// TIA Portal V17 program export: 0 tag tables, 0 data types, 0 data blocks, 2 code blocks (in call order from the OBs), 7 instance data blocks

ORGANIZATION_BLOCK "Main"   // OB1, LAD, ProgramCycle
TITLE = "Main Program Sweep (Cycle)"
{ S7_Optimized_Access := 'TRUE' }
VERSION : 0.1
// stored: AutoNumber true, IsIECCheckEnabled false, SetENOAutomatically false
   VAR_INPUT
      Initial_Call : Bool;   // Initial call of this OB
      Remanence : Bool;   // =True, if remanent data are available
   END_VAR
BEGIN

REGION Network 1
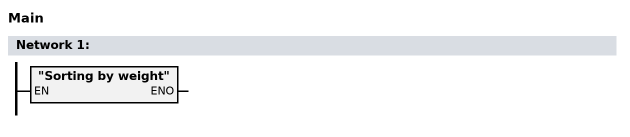
   RUNG wire#powerrail
      "Sorting by weight"()
   END_RUNG
   // the same network as SCL:
   "Sorting by weight"();
END_REGION
END_ORGANIZATION_BLOCK

FUNCTION "Sorting by weight" : Void
{ S7_Optimized_Access := 'TRUE' }
VERSION : 0.1

BEGIN
	IF "Start_PB" THEN
	    "MainConveyor" := TRUE;
	    "LeftConveyor" := TRUE;
	    "MiddleConveyor" := TRUE;
	    "RightConveyor" := TRUE;
	
	END_IF;
	
	
	"IEC_Timer_0_DB".TOF(IN:=NOT "Stop_Sensor",
	                     PT:=T#1S);
	"F_TRIG_DB"(CLK:="IEC_Timer_0_DB".Q);
	
	"IEC_Timer_0_DB_1".TOF(IN:=NOT "Stop_Sensor",
	                       PT:=T#3S);
	"F_TRIG_DB_1"(CLK:="IEC_Timer_0_DB_1".Q);
	
	
	IF "F_TRIG_DB".Q THEN
	    "ConveyorScale" := FALSE;
	ELSIF NOT "Stop_Sensor" THEN
	    "ConveyorScale" := TRUE;
	ELSIF "F_TRIG_DB_1".Q THEN
	    "ConveyorScale" := TRUE;
	END_IF;
	
	
	// Scaling of weight
	"Actual Weight":="ConveyorScaleWight"*2.0;
	
	
	//compare weight and respective data register
	IF NOT "ConveyorScale" AND "Actual Weight" >= 8.0 AND "Actual Weight" <= 8.2 THEN
	    "SortBIT" := 1;
	ELSIF NOT "ConveyorScale" AND "Actual Weight" >= 10.0 AND "Actual Weight" <= 10.2 THEN
	    "SortBIT" := 2;
	ELSIF NOT "ConveyorScale" AND "Actual Weight" > 15.0   THEN
	    "SortBIT" := 3;
	END_IF;
	
	
	// sort forward 10kg box
	IF "SortBIT"=2 THEN
	    "SortForword" := true;
	END_IF;
	
	// Reset forward sorting
	IF NOT "ExitSensorMiddle" THEN
	    "SortForword" := FALSE;
	    "SortLeft" := FALSE;
	    "SortRight" := FALSE;
	    "SortBIT" := 0;
	    "ConveyorScale" := FALSE;
	END_IF;
	
	
	// sort left 8kg box
	IF "SortBIT" = 1 THEN
	    "SortForword" := true;
	    "SortLeft" := true;
	END_IF;
	
	//reset left sorting
	IF NOT "ExitSensorLeft" THEN
	    "SortForword" := FALSE;
	    "SortLeft" := FALSE;
	    "SortRight" := FALSE;
	    "SortBIT" := 0;
	    "ConveyorScale" := 0;
	END_IF;
	
	
	// Sort right 15kg box
	IF "SortBIT" = 3 THEN
	    "SortForword" := true;
	    "SortRight" := true;
	END_IF;
	
	//reset right sorting 
	IF NOT "ExitSensorRight" THEN
	    "SortForword" := FALSE;
	    "SortLeft" := FALSE;
	    "SortRight" := FALSE;
	    "SortBIT" := 0;
	    "ConveyorScale" := 0;
	END_IF;
	
	
	// RESET ALL OUTPUT, MEMORY BIT , AND DATA REGISTER
	IF "Reset_PB" THEN
	    "Tag_3" := 0;
	    "Actual Weight" := 0;
	    "SortBIT" := 0;
	END_IF;
	
	// counting box
	"IEC_Counter_0_DB".CTU(CU:="ExitSensorLeft",
	                       PV:=100,
	                       CV=>"8KG_BoxCounter");
	
	"IEC_Counter_0_DB_1".CTU(CU:="ExitSensorMiddle",
	                         PV:=100,
	                         CV=>"10KG_BoxCounter");
	
	"IEC_Counter_0_DB_2".CTU(CU:="ExitSensorRight",
	                         PV:=100,
	                         CV=>"15KG_BoxCounter");
	
	
	
	
	
	
END_FUNCTION

DATA_BLOCK "F_TRIG_DB"   // DB2
// stored: AutoNumber true, DBAccessibleFromOPCUA true, DBAccessibleFromWebserver true, InstanceOfName F_TRIG, OfSystemLibElement F_TRIG, OfSystemLibVersion 1.0
"F_TRIG"
   // VAR_INPUT
   //    CLK : Bool;
   // END_VAR
   // VAR_OUTPUT
   //    Q : Bool;
   // END_VAR
   // VAR
   //    Stat_Bit : Bool;
   // END_VAR
BEGIN
END_DATA_BLOCK

DATA_BLOCK "F_TRIG_DB_1"   // DB4
// stored: AutoNumber true, DBAccessibleFromOPCUA true, DBAccessibleFromWebserver true, InstanceOfName F_TRIG, OfSystemLibElement F_TRIG, OfSystemLibVersion 1.0
"F_TRIG"
   // VAR_INPUT
   //    CLK : Bool;
   // END_VAR
   // VAR_OUTPUT
   //    Q : Bool;
   // END_VAR
   // VAR
   //    Stat_Bit : Bool;
   // END_VAR
BEGIN
END_DATA_BLOCK

DATA_BLOCK "IEC_Counter_0_DB"   // DB5
{ S7_Optimized_Access := 'TRUE' }
// stored: AutoNumber true, DBAccessibleFromOPCUA true, DBAccessibleFromWebserver true, InstanceOfName IEC_COUNTER, OfSystemLibElement IEC_COUNTER, OfSystemLibVersion 1.0
"IEC_COUNTER"
   // VAR RETAIN
   //    CU : Bool;
   //    CD : Bool;
   //    R : Bool;
   //    LD : Bool;
   //    QU : Bool;
   //    QD : Bool;
   //    PV : Int;
   //    CV : Int;
   // END_VAR
BEGIN
END_DATA_BLOCK

DATA_BLOCK "IEC_Counter_0_DB_1"   // DB6
{ S7_Optimized_Access := 'TRUE' }
// stored: AutoNumber true, DBAccessibleFromOPCUA true, DBAccessibleFromWebserver true, InstanceOfName IEC_COUNTER, OfSystemLibElement IEC_COUNTER, OfSystemLibVersion 1.0
"IEC_COUNTER"
   // VAR RETAIN
   //    CU : Bool;
   //    CD : Bool;
   //    R : Bool;
   //    LD : Bool;
   //    QU : Bool;
   //    QD : Bool;
   //    PV : Int;
   //    CV : Int;
   // END_VAR
BEGIN
END_DATA_BLOCK

DATA_BLOCK "IEC_Counter_0_DB_2"   // DB7
{ S7_Optimized_Access := 'TRUE' }
// stored: AutoNumber true, DBAccessibleFromOPCUA true, DBAccessibleFromWebserver true, InstanceOfName IEC_COUNTER, OfSystemLibElement IEC_COUNTER, OfSystemLibVersion 1.0
"IEC_COUNTER"
   // VAR RETAIN
   //    CU : Bool;
   //    CD : Bool;
   //    R : Bool;
   //    LD : Bool;
   //    QU : Bool;
   //    QD : Bool;
   //    PV : Int;
   //    CV : Int;
   // END_VAR
BEGIN
END_DATA_BLOCK

DATA_BLOCK "IEC_Timer_0_DB"   // DB1
{ S7_Optimized_Access := 'TRUE' }
// stored: AutoNumber true, DBAccessibleFromOPCUA true, DBAccessibleFromWebserver true, InstanceOfName IEC_TIMER, OfSystemLibElement IEC_TIMER, OfSystemLibVersion 1.0
"IEC_TIMER"
   // VAR
   //    PT : Time;
   //    ET { ExternalWritable := 'False'} : Time;
   //    IN : Bool;
   //    Q { ExternalWritable := 'False'} : Bool;
   // END_VAR
BEGIN
END_DATA_BLOCK

DATA_BLOCK "IEC_Timer_0_DB_1"   // DB3
{ S7_Optimized_Access := 'TRUE' }
// stored: AutoNumber true, DBAccessibleFromOPCUA true, DBAccessibleFromWebserver true, InstanceOfName IEC_TIMER, OfSystemLibElement IEC_TIMER, OfSystemLibVersion 1.0
"IEC_TIMER"
   // VAR
   //    PT : Time;
   //    ET { ExternalWritable := 'False'} : Time;
   //    IN : Bool;
   //    Q { ExternalWritable := 'False'} : Bool;
   // END_VAR
BEGIN
END_DATA_BLOCK
